Staubli VAL3: Light.pgx

public program Light(num x_nType (dimensions=1))
  local string l_sS
begin
  //对指示灯进行设置

  //0 红灯亮
  //1黄灯亮
  //2 绿灯亮


  //红
  call IOName(72,l_sS)
  dDio[l_sS]=(x_nType==0)
  //黄
  call IOName(73,l_sS)
  dDio[l_sS]=(x_nType==1)
  //绿
  call IOName(74,l_sS)
  dDio[l_sS]=(x_nType==2)
  //报警
  call IOName(75,l_sS)
  dDio[l_sS]=(x_nType==0)


end
